ABB RAPID module: Wobj_rfl_locexp_mdfplate2.mod

MODULE Wobj_rfl_locexp_mdfplate2
	! Points are read in order of declaration.
  ! Please do not change the order of points!

  LOCAL PERS robtarget pWobj_U_PointX1:=[[1797.468,-474.0795,-521.1123],[0.144962072372437,0.855986893177032,0.478719145059586,0.130768612027168],[-1,-2,2,0],[9E+09,9E+09,9E+09,9E+09,9E+09,9E+09]];
	LOCAL PERS robtarget pWobj_U_PointX2:=[[1717.137,-1079.697,-518.1675],[0.208680883049965,0.726086974143982,0.641686022281647,0.132246255874634],[-1,1,-1,0],[9E+09,9E+09,9E+09,9E+09,9E+09,9E+09]];
	LOCAL PERS robtarget pWobj_U_PointY1:=[[1799.409,-473.5343,398.8327],[0.208626046776772,0.726090967655182,0.641706228256226,0.132212713360786],[-1,-1,0,0],[9E+09,9E+09,9E+09,9E+09,9E+09,9E+09]];

ENDMODULE
